// TIA Portal V19 export
VAR_GLOBAL   // PLC tag table "Alarm_Tags"
   ACKPB AT %M3.3 : Bool;   // Alarm ACK
   RESETPB AT %M3.4 : Bool;   // Alarm Reset
   Alarm_1 AT %M3.5 : Bool;   // Alarm #No1
   Alarm1ACKED AT %M3.6 : Bool;   // Alarm #1 Acknowledged
   Alarm1LED AT %M3.7 : Bool;   // Alarm #1 LED
   StopBelt AT %M4.0 : Bool;   // E-Stop The Belt
   Alarm_2 AT %M4.1 : Bool;   // Alarm #No2
   Alarm2ACKED AT %M4.2 : Bool;   // Alarm #2 Acknowledged
   Alarm2LED AT %M4.3 : Bool;   // Alarm #2 LED
END_VAR
